Fanuc KAREL source: kx00003.KL

-- PROVISIONAL review KL for V770-1; original PC SHA256 204684e4850c355d4f85580620b6c0413c01cc2603b58d22efe1b695ed76df29
-- Incomplete behavior may be omitted. Consult companion uncertainty JSON. Do not deploy.
PROGRAM KX00003
%NOLOCKGROUP
VAR
  I : INTEGER
  J : INTEGER
  B : BOOLEAN
  F : FILE
  S : STRING[80]
-- UNRESOLVED_DECL P type=000102
BEGIN
  -- UNRESOLVED_PC offsets 5-32; opcodes 22,3F,3F,3D
  -- UNRESOLVED_PC offsets 37-65; opcodes 22,3F,9C,9C,37,9C,9C,37,2C
  -- UNRESOLVED_PC offsets 70-77; opcodes 22,39
  -- UNRESOLVED_PC offsets 82-86; opcodes 7F
END KX00003
